// TIA Portal project "testesBombaSSA" (V15)

(* hardware
DEVICE "S7-1200 station_1"  S7-1200 Station
   slot 0: "Rack_0"  S7-1200 Rack  Rack  V1.0
   slot 1: "PLC_1"  CPU 1217C DC/DC/DC  6ES7 217-1AG40-0XB0  V4.2
DEVICE "S7-1200 station_2"  S7-1200 Station
   slot 0: "Rack_0"  S7-1200 Rack  Rack  V1.0
   slot 1: "PLC_2"  CPU 1211C AC/DC/Rly  6ES7 211-1BD30-0XB0  V2.2
*)

// ===== PLC "PLC_1"  CPU 1217C DC/DC/DC =====

VAR_GLOBAL   // PLC tag table "Default tag table"
   "liga" AT %I0.0 : Bool;
   "manutencao" AT %I0.1 : Bool;
   "desliga" AT %I0.2 : Bool;
   "saida Disponivel" AT %Q0.4 : Bool;
   "saida Falha" AT %Q0.5 : Bool;
   "saida LocalRemoto" AT %Q1.0 : Bool;
   "saida Manutencao" AT %Q0.6 : Bool;
   "saida Recuperacao" AT %Q0.7 : Bool;
   "saida status Acionamento" AT %Q0.0 : Bool;
   "falha" AT %I0.3 : Bool;
   "memoria Liga" AT %M0.0 : Bool;
   "memoria falha" AT %M0.1 : Bool;
   "memoria desLiga" AT %M0.2 : Bool;
   "memoria manutencao" AT %M0.3 : Bool;
   "memoria local remoto" AT %M0.4 : Bool;
   "Tag_1" AT %I0.4 : Bool;
   "local remoto" AT %M0.4 : Bool;
   "remoto local" AT %M0.5 : Bool;
END_VAR

TYPE "PocosCaptacao"
   STRUCT
      iStatus : Int;
      bStatusAcionamento : Bool;
      bFalha : Bool;
      bDisponivel : Bool;
      bRecuperacao : Bool;
      bManutencao : Bool;
      bLocalRemoto : Bool;
      timeTotalizadoAcionamento : Time;
      timeRecuperacao : Time;
      dtUltimoAcionamento : DTL;
      dtUltimaManutencao : DTL;
      dtProximoAcionamento : DTL;
   END_STRUCT;
END_TYPE

DATA_BLOCK "Data_block_1"   // DB1
{ S7_Optimized_Access := 'TRUE' }
VERSION : 0.1
   VAR
      HoraAtual : DTL;
      poco01 : "PocosCaptacao";
   END_VAR
BEGIN
END_DATA_BLOCK

DATA_BLOCK "Interface_IHM"   // DB300
{ S7_Optimized_Access := 'TRUE' }
VERSION : 0.1
   VAR RETAIN
      poco01 : "PocosCaptacao";
   END_VAR
BEGIN
   poco01.bStatusAcionamento := false;
END_DATA_BLOCK

// folder: DB´s Pocos

DATA_BLOCK "FB_Pocos_DB_"   // DB201
{ S7_Optimized_Access := 'TRUE' }
VERSION : 0.1
// stored: InstanceOfName FB_Pocos
"FB_Pocos"
BEGIN
END_DATA_BLOCK

// folder: (top level)

FUNCTION_BLOCK "FB_Pocos"   // FB1, LAD
{ S7_Optimized_Access := 'TRUE' }
VERSION : 0.1
   VAR_IN_OUT
      info_poco : "PocosCaptacao";
   END_VAR
   VAR
      blnPocoLiberado : Bool;
      timeTempoUltimoAcionamento : Time;
      blnTmpPocoLiberado : Bool;
      blnTempAcionamento : Bool;
      blnTempAcionamentoOFF : Bool;
      blnTmpStatusPocoOFF : Bool;
      blnTempManutencao : Bool;
      timeInicioAcionamento : DTL;
      timeTempAcionamento : Time;
   END_VAR
   VAR_TEMP
      blnTmpStatusPoco : Bool;
   END_VAR
   VAR_TEMP   // added for the SCL form of the ladder/FBD networks
      _w1 : Bool;
      _w2 : Bool;
   END_VAR
BEGIN

REGION Network 1
   // Verifica se Poco esta Dentro do Intervalo de Recuperação
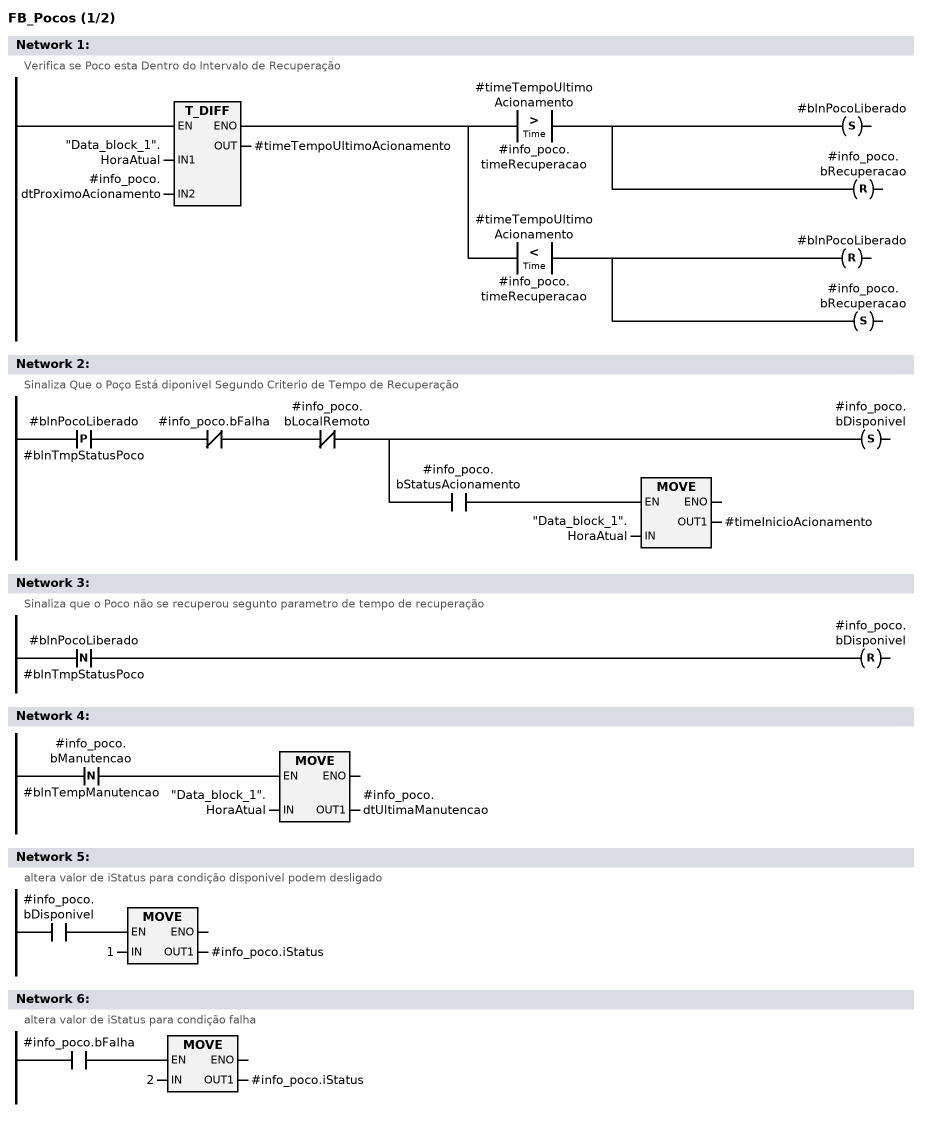
   // ENO of a box is taken as its EN; it also drops when the box reports an error
   #timeTempoUltimoAcionamento := T_DIFF(IN1 := "Data_block_1".HoraAtual,
                           IN2 := #info_poco.dtProximoAcionamento);
   IF #timeTempoUltimoAcionamento > #info_poco.timeRecuperacao THEN
       #blnPocoLiberado := TRUE;
       #info_poco.bRecuperacao := FALSE;
   END_IF;
   IF #timeTempoUltimoAcionamento < #info_poco.timeRecuperacao THEN
       #blnPocoLiberado := FALSE;
       #info_poco.bRecuperacao := TRUE;
   END_IF;
END_REGION

REGION Network 2
   // Sinaliza Que o Poço Está diponivel Segundo Criterio de Tempo de Recuperação
   RUNG wire#powerrail
      P_Contact(operand := #blnPocoLiberado, bit := #blnTmpStatusPoco)
      I_Contact( #info_poco.bFalha )
      I_Contact( #info_poco.bLocalRemoto )
      wire#w1
      S_Coil( #info_poco.bDisponivel )
   END_RUNG
   RUNG wire#w1
      Contact( #info_poco.bStatusAcionamento )
      Move(in := "Data_block_1".HoraAtual, out1 => #timeInicioAcionamento)
   END_RUNG
   // the same network as SCL:
   #_w1 := #blnPocoLiberado AND NOT #blnTmpStatusPoco;   // rising edge of #blnPocoLiberado
   #blnTmpStatusPoco := #blnPocoLiberado;
   #_w2 := #_w1 AND NOT #info_poco.bFalha AND NOT #info_poco.bLocalRemoto;
   IF #_w2 THEN #info_poco.bDisponivel := TRUE; END_IF;
   IF #_w2 AND #info_poco.bStatusAcionamento THEN #timeInicioAcionamento := "Data_block_1".HoraAtual; END_IF;
END_REGION

REGION Network 3
   // Sinaliza que o Poco não se recuperou segunto parametro de tempo de recuperação
   RUNG wire#powerrail
      N_Contact(operand := #blnPocoLiberado, bit := #blnTmpStatusPoco)
      R_Coil( #info_poco.bDisponivel )
   END_RUNG
   // the same network as SCL:
   #_w1 := NOT #blnPocoLiberado AND #blnTmpStatusPoco;   // falling edge of #blnPocoLiberado
   #blnTmpStatusPoco := #blnPocoLiberado;
   IF #_w1 THEN #info_poco.bDisponivel := FALSE; END_IF;
END_REGION

REGION Network 4
   RUNG wire#powerrail
      N_Contact(operand := #info_poco.bManutencao, bit := #blnTempManutencao)
      Move(in := "Data_block_1".HoraAtual, out1 => #info_poco.dtUltimaManutencao)
   END_RUNG
   // the same network as SCL:
   #_w1 := NOT #info_poco.bManutencao AND #blnTempManutencao;   // falling edge of #info_poco.bManutencao
   #blnTempManutencao := #info_poco.bManutencao;
   IF #_w1 THEN #info_poco.dtUltimaManutencao := "Data_block_1".HoraAtual; END_IF;
END_REGION

REGION Network 5
   // altera valor de iStatus para condição disponivel podem desligado
   RUNG wire#powerrail
      Contact( #info_poco.bDisponivel )
      Move(in := 1, out1 => #info_poco.iStatus)
   END_RUNG
   // the same network as SCL:
   IF #info_poco.bDisponivel THEN #info_poco.iStatus := 1; END_IF;
END_REGION

REGION Network 6
   // altera valor de iStatus para condição falha
   RUNG wire#powerrail
      Contact( #info_poco.bFalha )
      Move(in := 2, out1 => #info_poco.iStatus)
   END_RUNG
   // the same network as SCL:
   IF #info_poco.bFalha THEN #info_poco.iStatus := 2; END_IF;
END_REGION

REGION Network 7
   // altera valor de iStatus para condição manutenção
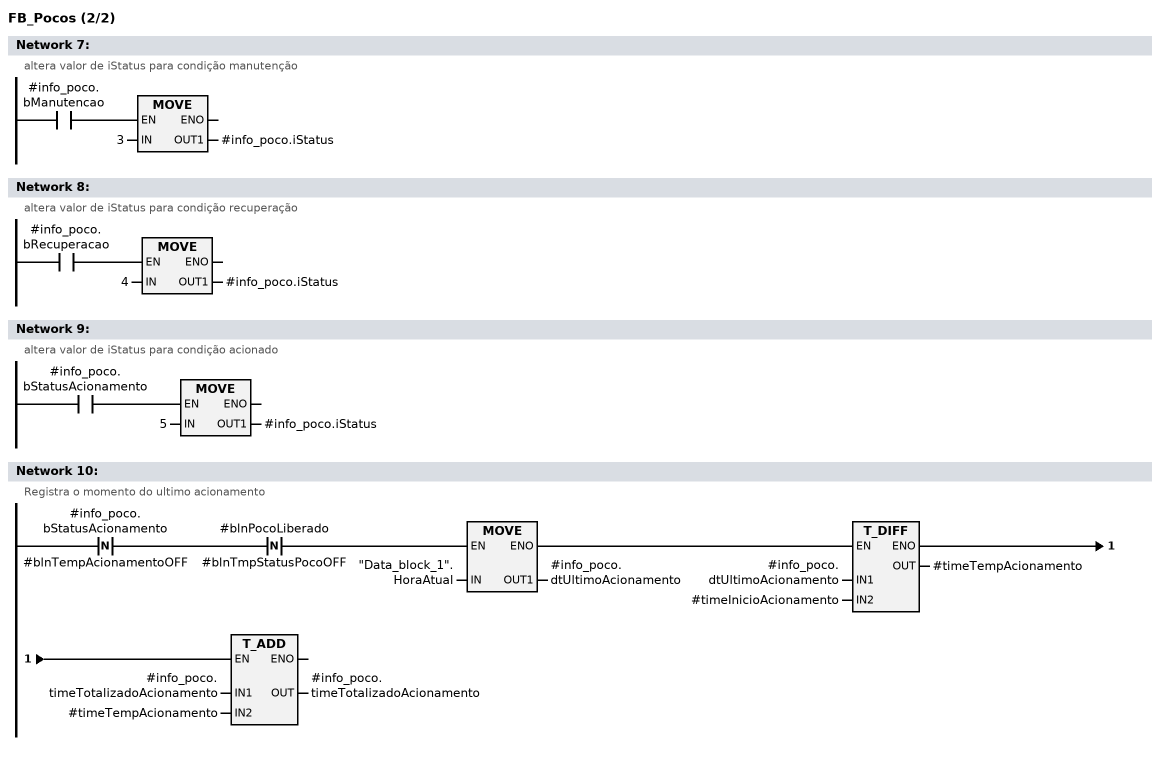
   RUNG wire#powerrail
      Contact( #info_poco.bManutencao )
      Move(in := 3, out1 => #info_poco.iStatus)
   END_RUNG
   // the same network as SCL:
   IF #info_poco.bManutencao THEN #info_poco.iStatus := 3; END_IF;
END_REGION

REGION Network 8
   // altera valor de iStatus para condição recuperação
   RUNG wire#powerrail
      Contact( #info_poco.bRecuperacao )
      Move(in := 4, out1 => #info_poco.iStatus)
   END_RUNG
   // the same network as SCL:
   IF #info_poco.bRecuperacao THEN #info_poco.iStatus := 4; END_IF;
END_REGION

REGION Network 9
   // altera valor de iStatus para condição acionado
   RUNG wire#powerrail
      Contact( #info_poco.bStatusAcionamento )
      Move(in := 5, out1 => #info_poco.iStatus)
   END_RUNG
   // the same network as SCL:
   IF #info_poco.bStatusAcionamento THEN #info_poco.iStatus := 5; END_IF;
END_REGION

REGION Network 10
   // Registra o momento do ultimo acionamento
   // ENO of a box is taken as its EN; it also drops when the box reports an error
   #_w1 := NOT #info_poco.bStatusAcionamento AND #blnTempAcionamentoOFF;   // falling edge of #info_poco.bStatusAcionamento
   #blnTempAcionamentoOFF := #info_poco.bStatusAcionamento;
   #_w2 := #_w1 AND NOT #blnPocoLiberado AND #blnTmpStatusPocoOFF;   // falling edge of #blnPocoLiberado
   #blnTmpStatusPocoOFF := #blnPocoLiberado;
   IF #_w2 THEN
       #info_poco.dtUltimoAcionamento := "Data_block_1".HoraAtual;
       #timeTempAcionamento := T_DIFF(IN1 := #info_poco.dtUltimoAcionamento, IN2 := #timeInicioAcionamento);
       #info_poco.timeTotalizadoAcionamento := T_ADD(IN1 := #info_poco.timeTotalizadoAcionamento,
                               IN2 := #timeTempAcionamento);
   END_IF;
END_REGION
END_FUNCTION_BLOCK

FUNCTION "interface Factoryoi" : Void   // FC1, LAD
{ S7_Optimized_Access := 'TRUE' }
VERSION : 0.1
   VAR_TEMP
      Temp_1 : Array[0..1] of Bool;
   END_VAR
   VAR_TEMP   // added for the SCL form of the ladder/FBD networks
      _w1 : Bool;
   END_VAR
BEGIN

REGION Network 1
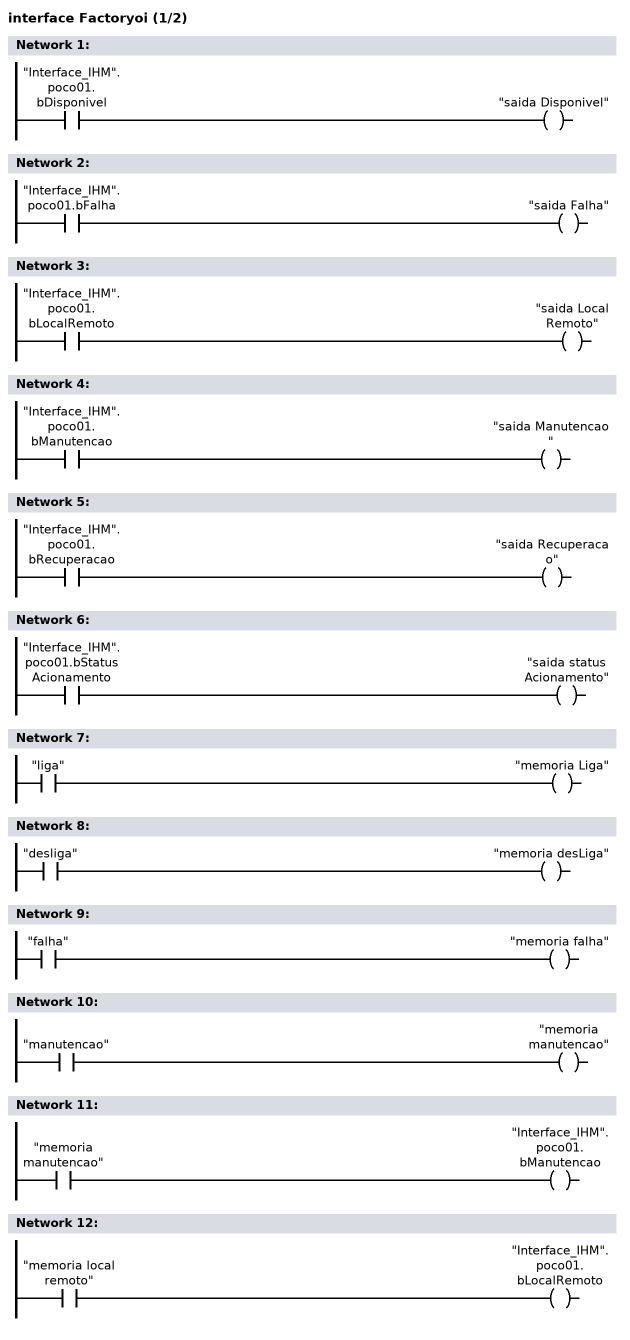
   RUNG wire#powerrail
      Contact( "Interface_IHM".poco01.bDisponivel )
      Coil( "saida Disponivel" )
   END_RUNG
   // the same network as SCL:
   "saida Disponivel" := "Interface_IHM".poco01.bDisponivel;
END_REGION

REGION Network 2
   RUNG wire#powerrail
      Contact( "Interface_IHM".poco01.bFalha )
      Coil( "saida Falha" )
   END_RUNG
   // the same network as SCL:
   "saida Falha" := "Interface_IHM".poco01.bFalha;
END_REGION

REGION Network 3
   RUNG wire#powerrail
      Contact( "Interface_IHM".poco01.bLocalRemoto )
      Coil( "saida LocalRemoto" )
   END_RUNG
   // the same network as SCL:
   "saida LocalRemoto" := "Interface_IHM".poco01.bLocalRemoto;
END_REGION

REGION Network 4
   RUNG wire#powerrail
      Contact( "Interface_IHM".poco01.bManutencao )
      Coil( "saida Manutencao" )
   END_RUNG
   // the same network as SCL:
   "saida Manutencao" := "Interface_IHM".poco01.bManutencao;
END_REGION

REGION Network 5
   RUNG wire#powerrail
      Contact( "Interface_IHM".poco01.bRecuperacao )
      Coil( "saida Recuperacao" )
   END_RUNG
   // the same network as SCL:
   "saida Recuperacao" := "Interface_IHM".poco01.bRecuperacao;
END_REGION

REGION Network 6
   RUNG wire#powerrail
      Contact( "Interface_IHM".poco01.bStatusAcionamento )
      Coil( "saida status Acionamento" )
   END_RUNG
   // the same network as SCL:
   "saida status Acionamento" := "Interface_IHM".poco01.bStatusAcionamento;
END_REGION

REGION Network 7
   RUNG wire#powerrail
      Contact( "liga" )
      Coil( "memoria Liga" )
   END_RUNG
   // the same network as SCL:
   "memoria Liga" := "liga";
END_REGION

REGION Network 8
   RUNG wire#powerrail
      Contact( "desliga" )
      Coil( "memoria desLiga" )
   END_RUNG
   // the same network as SCL:
   "memoria desLiga" := "desliga";
END_REGION

REGION Network 9
   RUNG wire#powerrail
      Contact( "falha" )
      Coil( "memoria falha" )
   END_RUNG
   // the same network as SCL:
   "memoria falha" := "falha";
END_REGION

REGION Network 10
   RUNG wire#powerrail
      Contact( "manutencao" )
      Coil( "memoria manutencao" )
   END_RUNG
   // the same network as SCL:
   "memoria manutencao" := "manutencao";
END_REGION

REGION Network 11
   RUNG wire#powerrail
      Contact( "memoria manutencao" )
      Coil( "Interface_IHM".poco01.bManutencao )
   END_RUNG
   // the same network as SCL:
   "Interface_IHM".poco01.bManutencao := "memoria manutencao";
END_REGION

REGION Network 12
   RUNG wire#powerrail
      Contact( "memoria local remoto" )
      Coil( "Interface_IHM".poco01.bLocalRemoto )
   END_RUNG
   // the same network as SCL:
   "Interface_IHM".poco01.bLocalRemoto := "memoria local remoto";
END_REGION

REGION Network 13
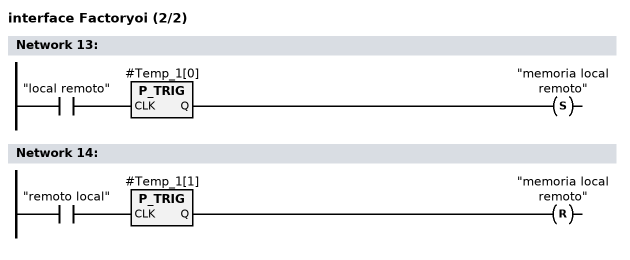
   RUNG wire#powerrail
      Contact( "local remoto" )
      P_Trig( #Temp_1[0] )
      S_Coil( "memoria local remoto" )
   END_RUNG
   // the same network as SCL:
   #_w1 := "local remoto" AND NOT #Temp_1[0];   // rising edge
   #Temp_1[0] := "local remoto";
   IF #_w1 THEN "memoria local remoto" := TRUE; END_IF;
END_REGION

REGION Network 14
   RUNG wire#powerrail
      Contact( "remoto local" )
      P_Trig( #Temp_1[1] )
      R_Coil( "memoria local remoto" )
   END_RUNG
   // the same network as SCL:
   #_w1 := "remoto local" AND NOT #Temp_1[1];   // rising edge
   #Temp_1[1] := "remoto local";
   IF #_w1 THEN "memoria local remoto" := FALSE; END_IF;
END_REGION
END_FUNCTION

FUNCTION "Acionamento _Pocos" : Void   // FC100, LAD
{ S7_Optimized_Access := 'TRUE' }
VERSION : 0.1
BEGIN

REGION Network 1
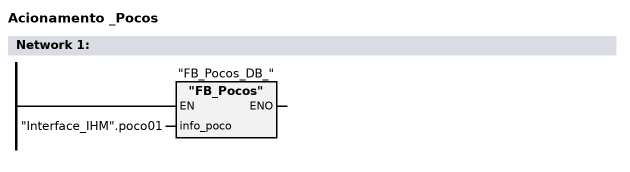
   RUNG wire#powerrail
      "FB_Pocos_DB_"(info_poco := "Interface_IHM".poco01)
   END_RUNG
   // the same network as SCL:
   "FB_Pocos_DB_"(info_poco := "Interface_IHM".poco01);   // "FB_Pocos"
END_REGION
END_FUNCTION

FUNCTION "MHJ-PLC-Lab-Function-S71200" : Void   // FC9000, SCL
{ S7_Optimized_Access := 'TRUE' }
VERSION : 0.1
   VAR_TEMP
      rdTimeReturn : Int;
      outputTime : DTL;
      SyncVal : Byte;
      forVal : Int;
      forVal_2 : Int;
      Value : Byte;
   END_VAR
   VAR CONSTANT
      CompVal : Byte := 16#34;
      Value_01 : Byte := 16#11;
      Value_01_DW : DWord := 16#A165_D992;
      Value_02_DW : DWord := 16#58BE_4401;
   END_VAR
BEGIN

   #Value:=PEEK(area := 16#82,
        dbNumber := 0,
        byteOffset := 511);
   #Value := #Value + 1;

   POKE(area := 16#82,
        dbNumber := 0,
        byteOffset := 511,
        value := #Value);

   POKE(area:=16#81,
        dbNumber:=0,
        byteOffset:=1016,
        value:=#Value_01_DW);
   POKE(area := 16#81,
        dbNumber := 0,
        byteOffset := 1020,
        value := #Value_02_DW);

   POKE(area := 16#81,
        dbNumber := 0,
        byteOffset := 511,
        value := B#16#00);

   FOR #forVal := 0 TO 120 DO
       FOR #forVal_2:=0 TO 10 DO
           #rdTimeReturn:=RD_SYS_T(#outputTime);
           #rdTimeReturn := WR_SYS_T(#outputTime);
           #rdTimeReturn := RD_SYS_T(#outputTime);
           #rdTimeReturn := WR_SYS_T(#outputTime);
       END_FOR;
       #SyncVal:= PEEK(area := 16#81,
                      dbNumber := 0,
                      byteOffset := 511);
       IF #SyncVal = #CompVal THEN
          GOTO M_1;
       END_IF;
   END_FOR;
   RETURN;

   M_1:
   POKE(area := 16#81,
        dbNumber := 0,
        byteOffset := 511,
        value := B#16#0);
END_FUNCTION

ORGANIZATION_BLOCK "Main"   // OB1, LAD, ProgramCycle
TITLE = "Main Program Sweep (Cycle)"
{ S7_Optimized_Access := 'TRUE' }
VERSION : 0.1
   VAR_INPUT
      Initial_Call : Bool;   // Initial call of this OB
      Remanence : Bool;   // =True, if remanent data are available
   END_VAR
   VAR_TEMP
      temp : Int;
      teste01 : Bool;
      teste02 : Bool;
   END_VAR
BEGIN

REGION Network 1
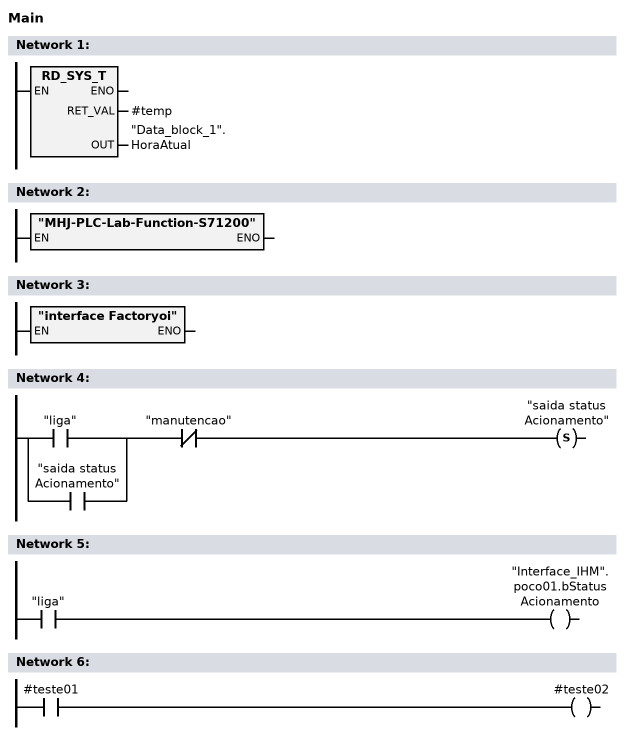
   #temp := RD_SYS_T(OUT => "Data_block_1".HoraAtual);
END_REGION

REGION Network 2
   RUNG wire#powerrail
      "MHJ-PLC-Lab-Function-S71200"()
   END_RUNG
   // the same network as SCL:
   "MHJ-PLC-Lab-Function-S71200"();
END_REGION

REGION Network 3
   RUNG wire#powerrail
      "interface Factoryoi"()
   END_RUNG
   // the same network as SCL:
   "interface Factoryoi"();
END_REGION

REGION Network 4
   RUNG wire#powerrail
      Contact( "liga" )
      wire#w1
      I_Contact( "manutencao" )
      S_Coil( "saida status Acionamento" )
   END_RUNG
   RUNG wire#powerrail
      Contact( "saida status Acionamento" )
   END_RUNG wire#w1
   // the same network as SCL:
   IF ("liga" OR "saida status Acionamento") AND NOT "manutencao" THEN
       "saida status Acionamento" := TRUE;
   END_IF;
END_REGION

REGION Network 5
   RUNG wire#powerrail
      Contact( "liga" )
      Coil( "Interface_IHM".poco01.bStatusAcionamento )
   END_RUNG
   // the same network as SCL:
   "Interface_IHM".poco01.bStatusAcionamento := "liga";
END_REGION

REGION Network 6
   RUNG wire#powerrail
      Contact( #teste01 )
      Coil( #teste02 )
   END_RUNG
   // the same network as SCL:
   #teste02 := #teste01;
END_REGION
END_ORGANIZATION_BLOCK

// ===== PLC "PLC_2"  CPU 1211C AC/DC/Rly =====

ORGANIZATION_BLOCK "Main"   // OB1, LAD, ProgramCycle
TITLE = "Main Program Sweep (Cycle)"
{ S7_Optimized_Access := 'TRUE' }
VERSION : 0.1
BEGIN
END_ORGANIZATION_BLOCK